FUNCTION BoolArrayToInteger : LINT;
VAR_IN_OUT
	arr : ARRAY[*] OF BOOL;
END_VAR
VAR
	i : DINT;
	j : DINT;
END_VAR

BoolArrayToInteger := 0;
(*
FOR i:=LOWER_BOUND(arr, 1) TO UPPER_BOUND(arr, 1) BY 1 DO
	
	IF j < SIZEOF(BoolArrayToInteger) * 8 THEN
		BoolArrayToInteger := SHL(BoolArrayToInteger, 1);
		BoolArrayToInteger.0 := arr[i];
	END_IF
	
END_FOR
*)
//iterate backwards
FOR i:=UPPER_BOUND(arr, 1) TO LOWER_BOUND(arr, 1) BY -1 DO
	
	IF j < SIZEOF(BoolArrayToInteger) * 8 THEN
		BoolArrayToInteger := SHL(BoolArrayToInteger, 1);
		BoolArrayToInteger.0 := arr[i];
	END_IF
	
END_FOR

END_FUNCTION

(* stored: Version 1.1.0.1, ProductVersion 3.1.4024.11
   POU BoolArrayToInteger: Id {125fe3f0-424f-4fff-9453-ca039cf450f3}, SpecialFunc None *)
